# EPICS substitutions: ucmApp/Db/undulator/xxUndulatorDispAlarmSum.substitutions
file xxUndulatorDispAlarmSum.template{
  pattern { motor  }
          { CM1 }
          { CM2 }
          { CM3 }
          { CM4 }
          { CM5 }
          { TM1 }
          { TM2 }
}
